% RSLogix 500 project I2P Job 16 - Myah.RSS, saved by version 10.00.00.00 %
PROJECT "UNTITLED"    % processor: Bul.1763 MicroLogix 1100 Series B %

PROGRAM FILES
  LAD 2   5 rungs

DATA FILES
  O0 OUTPUT  4 elements
  I1 INPUT  6 elements
  S2 STATUS  66 elements
  B3 BINARY  1 elements
  T4 TIMER  1 elements
  C5 COUNTER  1 elements
  R6 CONTROL  1 elements
  N7 INTEGER  1 elements
  F8 FLOAT  1 elements

LADDER 2
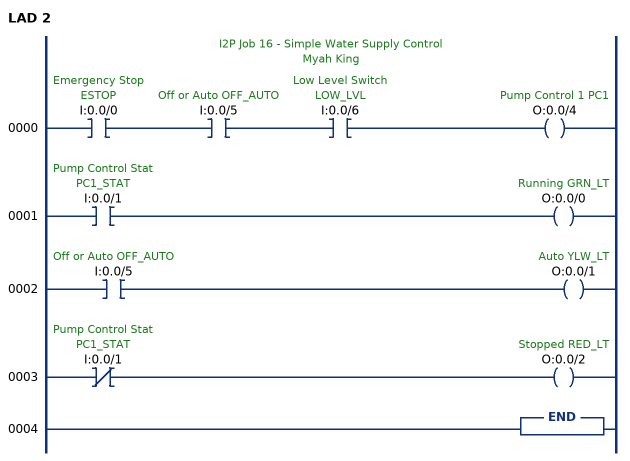
% Rung: 0 %
% I2P Job 16 - Simple Water Supply Control
% Myah King %
SOR XIC I:0.0/0 XIC I:0.0/5 XIC I:0.0/6 OTE O:0.0/4 EOR
%   I:0.0/0  ESTOP  "Emergency Stop" %
%   I:0.0/5  OFF_AUTO  "Off or Auto" %
%   I:0.0/6  LOW_LVL  "Low Level Switch" %
%   O:0.0/4  PC1  "Pump Control 1" %
% Rung: 1 %
SOR XIC I:0.0/1 OTE O:0.0/0 EOR
%   I:0.0/1  PC1_STAT  "Pump Control Stat" %
%   O:0.0/0  GRN_LT  "Running" %
% Rung: 2 %
SOR XIC I:0.0/5 OTE O:0.0/1 EOR
%   I:0.0/5  OFF_AUTO  "Off or Auto" %
%   O:0.0/1  YLW_LT  "Auto" %
% Rung: 3 %  % edit flag set %
SOR XIO I:0.0/1 OTE O:0.0/2 EOR
%   I:0.0/1  PC1_STAT  "Pump Control Stat" %
%   O:0.0/2  RED_LT  "Stopped" %
% Rung: 4 %
SOR END EOR
